// Mitsubishi GX Works2 project: demoDanNhan   PLC: FX3G

PROGRAM MAIN
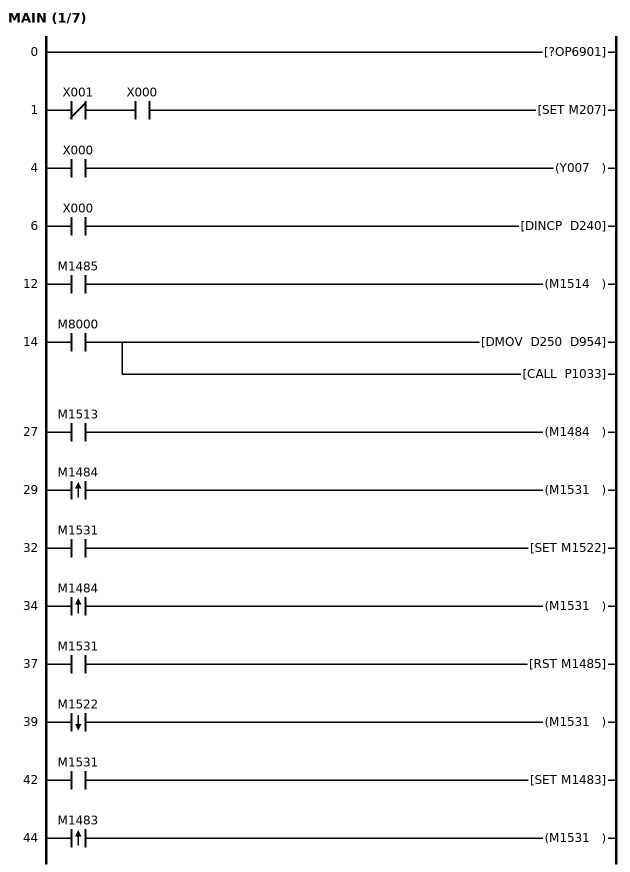
0     ?OP6901
1     LDI     X001
      AND     X000
      SET     M207
4     LD      X000
      OUT     Y007
6     LD      X000
      DINCP   D240
12    LD      M1485
      OUT     M1514
14    LD      M8000
      DMOV    D250 D954
      CALL    P1033
27    LD      M1513
      OUT     M1484
29    LDP     M1484
      OUT     M1531
32    LD      M1531
      SET     M1522
34    LDP     M1484
      OUT     M1531
37    LD      M1531
      RST     M1485
39    LDF     M1522
      OUT     M1531
42    LD      M1531
      SET     M1483
44    LDP     M1483
      OUT     M1531
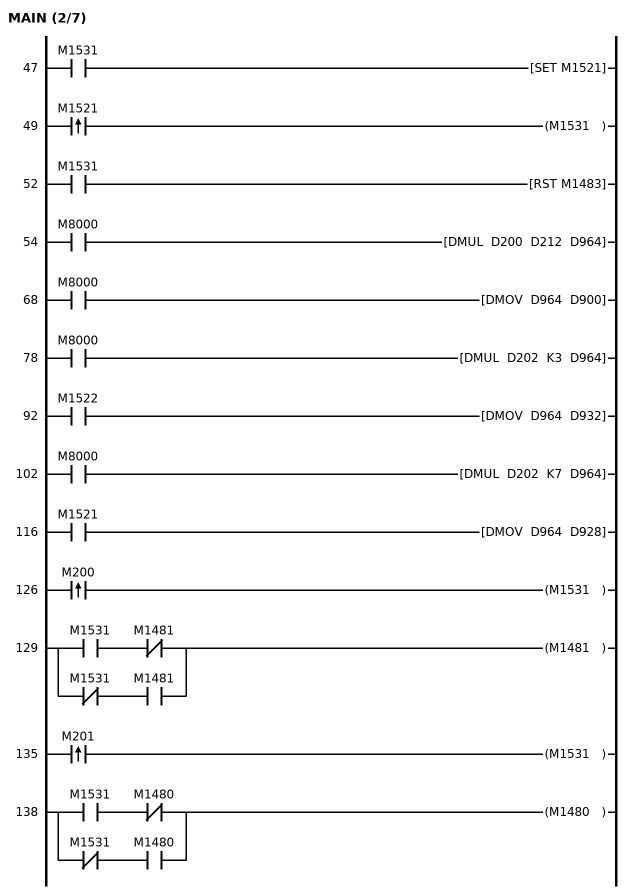
47    LD      M1531
      SET     M1521
49    LDP     M1521
      OUT     M1531
52    LD      M1531
      RST     M1483
54    LD      M8000
      DMUL    D200 D212 D964
68    LD      M8000
      DMOV    D964 D900
78    LD      M8000
      DMUL    D202 K3 D964
92    LD      M1522
      DMOV    D964 D932
102   LD      M8000
      DMUL    D202 K7 D964
116   LD      M1521
      DMOV    D964 D928
126   LDP     M200
      OUT     M1531
129   LD      M1531
      ANI     M1481
      LDI     M1531
      AND     M1481
      ORB
      OUT     M1481
135   LDP     M201
      OUT     M1531
138   LD      M1531
      ANI     M1480
      LDI     M1531
      AND     M1480
      ORB
      OUT     M1480
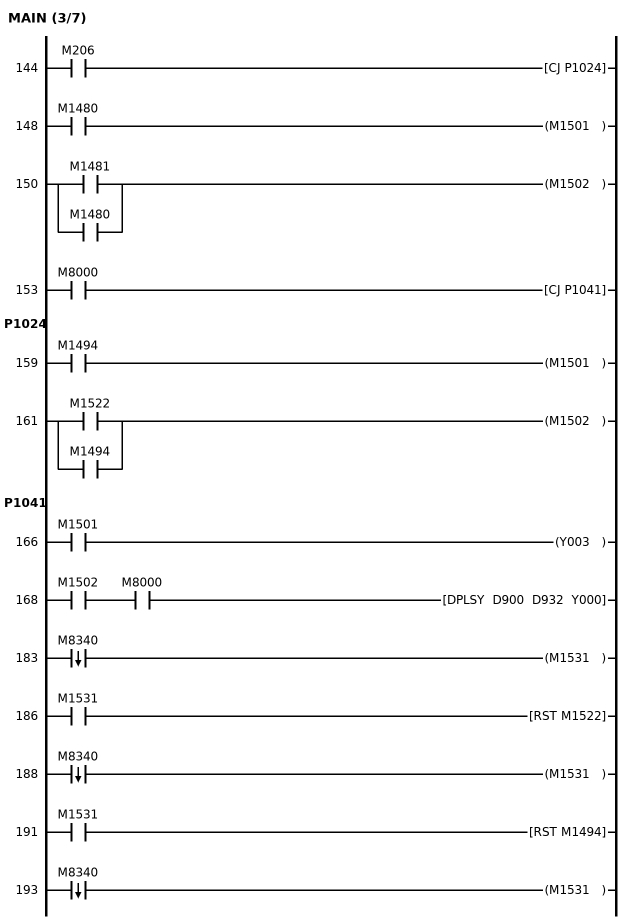
144   LD      M206
      CJ      P1024
148   LD      M1480
      OUT     M1501
150   LD      M1481
      OR      M1480
      OUT     M1502
153   LD      M8000
      CJ      P1041
      P1024
159   LD      M1494
      OUT     M1501
161   LD      M1522
      OR      M1494
      OUT     M1502
      P1041
166   LD      M1501
      OUT     Y003
168   LD      M1502
      AND     M8000
      DPLSY   D900 D932 Y000
183   LDF     M8340
      OUT     M1531
186   LD      M1531
      RST     M1522
188   LDF     M8340
      OUT     M1531
191   LD      M1531
      RST     M1494
193   LDF     M8340
      OUT     M1531
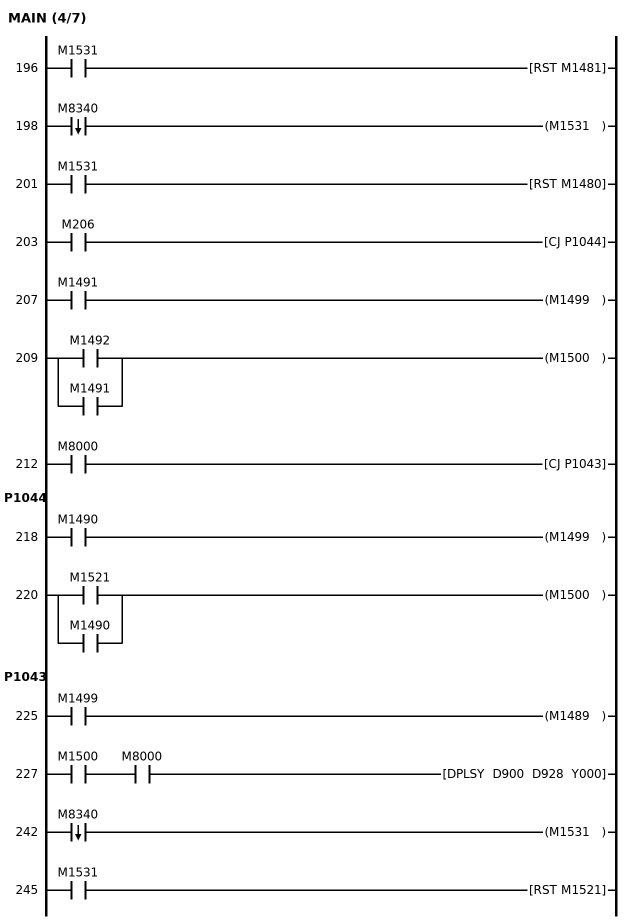
196   LD      M1531
      RST     M1481
198   LDF     M8340
      OUT     M1531
201   LD      M1531
      RST     M1480
203   LD      M206
      CJ      P1044
207   LD      M1491
      OUT     M1499
209   LD      M1492
      OR      M1491
      OUT     M1500
212   LD      M8000
      CJ      P1043
      P1044
218   LD      M1490
      OUT     M1499
220   LD      M1521
      OR      M1490
      OUT     M1500
      P1043
225   LD      M1499
      OUT     M1489
227   LD      M1500
      AND     M8000
      DPLSY   D900 D928 Y000
242   LDF     M8340
      OUT     M1531
245   LD      M1531
      RST     M1521
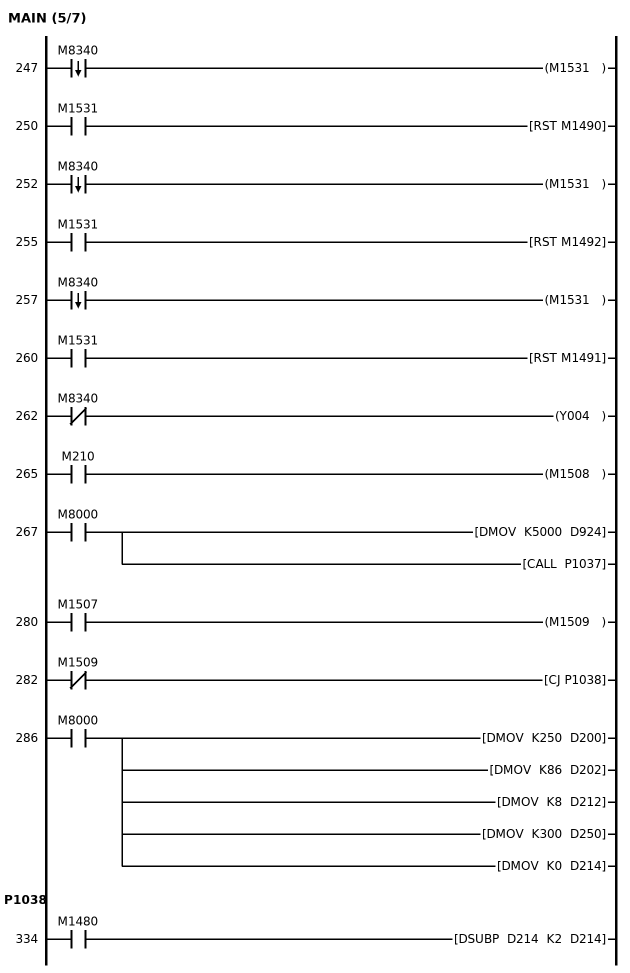
247   LDF     M8340
      OUT     M1531
250   LD      M1531
      RST     M1490
252   LDF     M8340
      OUT     M1531
255   LD      M1531
      RST     M1492
257   LDF     M8340
      OUT     M1531
260   LD      M1531
      RST     M1491
262   LDI     M8340
      OUT     Y004
265   LD      M210
      OUT     M1508
267   LD      M8000
      DMOV    K5000 D924
      CALL    P1037
280   LD      M1507
      OUT     M1509
282   LDI     M1509
      CJ      P1038
286   LD      M8000
      DMOV    K250 D200
      DMOV    K86 D202
      DMOV    K8 D212
      DMOV    K300 D250
      DMOV    K0 D214
      P1038
334   LD      M1480
      DSUBP   D214 K2 D214
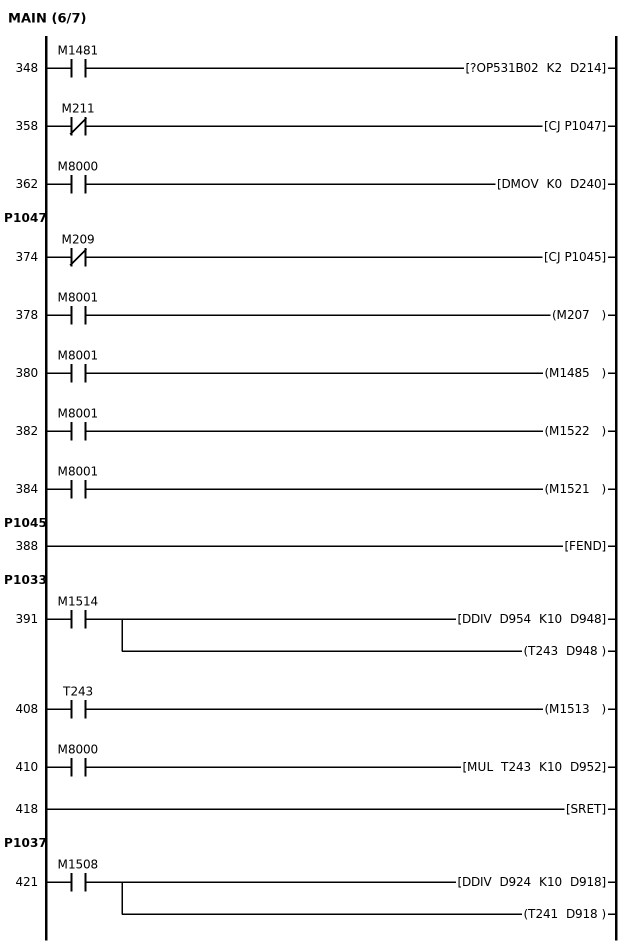
348   LD      M1481
      ?OP531B02 K2 D214
358   LDI     M211
      CJ      P1047
362   LD      M8000
      DMOV    K0 D240
      P1047
374   LDI     M209
      CJ      P1045
378   LD      M8001
      OUT     M207
380   LD      M8001
      OUT     M1485
382   LD      M8001
      OUT     M1522
384   LD      M8001
      OUT     M1521
      P1045
388   FEND
      P1033
391   LD      M1514
      DDIV    D954 K10 D948
      OUT     T243 D948
408   LD      T243
      OUT     M1513
410   LD      M8000
      MUL     T243 K10 D952
418   SRET
      P1037
421   LD      M1508
      DDIV    D924 K10 D918
      OUT     T241 D918
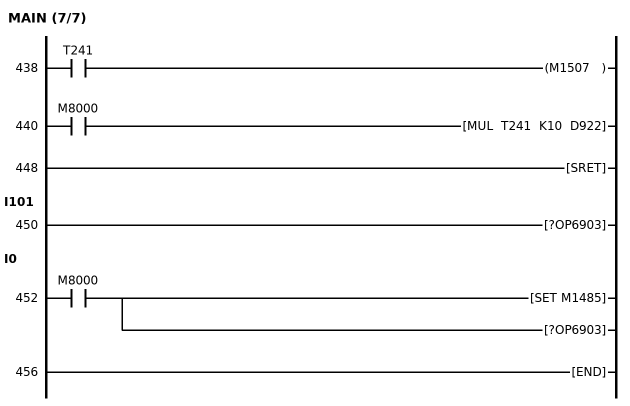
438   LD      T241
      OUT     M1507
440   LD      M8000
      MUL     T241 K10 D922
448   SRET
      I101
450   ?OP6903
      I0
452   LD      M8000
      SET     M1485
      ?OP6903
456   END
END_PROGRAM
